FUNCTION_BLOCK Filling_control
  (* Standard: 61499-2 *)
  (* Version 0.1, 2015-00-13, Th?o, PC_THEO *)
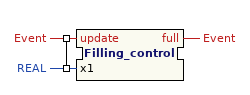
  EVENT_INPUT
    update WITH x1;
  END_EVENT
  EVENT_OUTPUT
    full;
  END_EVENT
  VAR_INPUT
    x1 : REAL;
  END_VAR
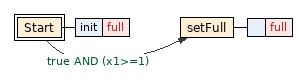
  EC_STATES
    Start : init -> full;
    setFull : -> full;
  END_STATES
  EC_TRANSITIONS
    Start TO setFull := true AND (x1>=1);
  END_TRANSITIONS
  ALGORITHM init IN C:
me->x1=0.05;
  END_ALGORITHM
END_FUNCTION_BLOCK
